Staubli VAL3: goTo.pgx

public program goTo(tool x_tTool, mdesc x_mDesc, num x_nMoveType, bool& x_bUnreached[], num x_nIndex)
  local point l_pTrsf
  local bool l_bInside
  local tool l_tTool
  local point l_pHere
  local string l_sMessage
  local num l_nSize
  local num i
  local mdesc l_mSpeed
  local joint l_jJoint
  local point l_pPoint[2]
  local bool l_bUnreach
begin
  // get the moveType
  call findMove(x_nIndex,x_tTool,x_nMoveType)
  if isEmpty()
    // get the POINT
    call getPoint(l_pPoint,false,x_nIndex)
    pToGo=l_pPoint
    pToGo[1]=l_pPoint[1]
    l_pHere=here(x_tTool,pEditPoint.fFrame)
    // step by step motion
    if x_nMoveType==0
      // or is not in range
      movej(pToGo,x_tTool,x_mDesc)
    elseIf x_nMoveType==1
      movel(pToGo,x_tTool,x_mDesc)
    elseIf x_nMoveType>2
      // inside the trajectory
      // take the percentage arcInterpo
      call getPoint(l_pPoint,false,x_nIndex-1)
      call isReachable(pToGo,x_tTool,l_bUnreach)
      if !l_bUnreach and pointToJoint(x_tTool,herej(),l_pPoint,l_jJoint)
        pToGo[1].trsf=interpolateC(position(l_pPoint,pEditPoint.fFrame),pToGo[1].trsf,pToGo.trsf,(1-(2-x_nMoveType))/2)
      endIf
    elseIf x_nMoveType<=-2
      // move circular backward
      call getPoint(l_pPoint,false,x_nIndex+1)
      call isReachable(l_pPoint,x_tTool,l_bUnreach)
      if !l_bUnreach
        // look for percentage value need
        if x_nMoveType==-2
          pToGo[1].trsf=position(l_pPoint[1],pEditPoint.fFrame)
        else
          pToGo[1].trsf=interpolateC(pToGo.trsf,position(l_pPoint[1],pEditPoint.fFrame),position(l_pPoint,pEditPoint.fFrame),(abs(x_nMoveType+2))/2)
        endIf
      endIf
    endIf
    if l_bUnreach
      // get the message point is not reachable
      call language:message(l_sMessage,-5)
      call use:type(0,12,"!!! "+l_sMessage)
    elseIf x_nMoveType!=0 and x_nMoveType!=1
      // CIRCULAR MOVE
      movec(pToGo[1],pToGo,x_tTool,x_mDesc)
    endIf
  endIf
end
